FUNCTION_BLOCK FB_TurboExtLogic
VAR_IN_OUT
	Turbo		:	ST_AgilentPTM;
END_VAR
VAR_INPUT
	BackingGauge:	ST_VG;
	InletGauge	:	ST_VG;
	VentValve	:	ST_VCC_NO;
	ScrollPump	:	ST_RoughPump;
END_VAR
VAR_OUTPUT
END_VAR
VAR
END_VAR

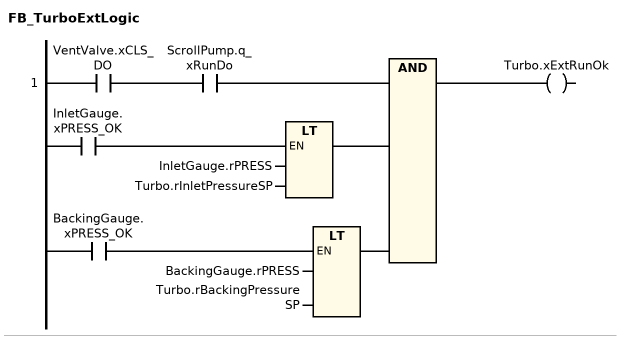
// NETWORK 1
Turbo.xExtRunOk := (VentValve.xCLS_DO AND ScrollPump.q_xRunDo) AND (InletGauge.xPRESS_OK AND InletGauge.rPRESS < Turbo.rInletPressureSP) AND (BackingGauge.xPRESS_OK AND BackingGauge.rPRESS < Turbo.rBackingPressureSP);

END_FUNCTION_BLOCK

(* stored: Version 1.1.0.1, ProductVersion 3.1.4020.12
   POU FB_TurboExtLogic: Id {1c568a9f-ee7d-4da0-9111-bdd0aa6cb7c8}, SpecialFunc None *)
